RoboDK station: Robot_2TCP.rdk

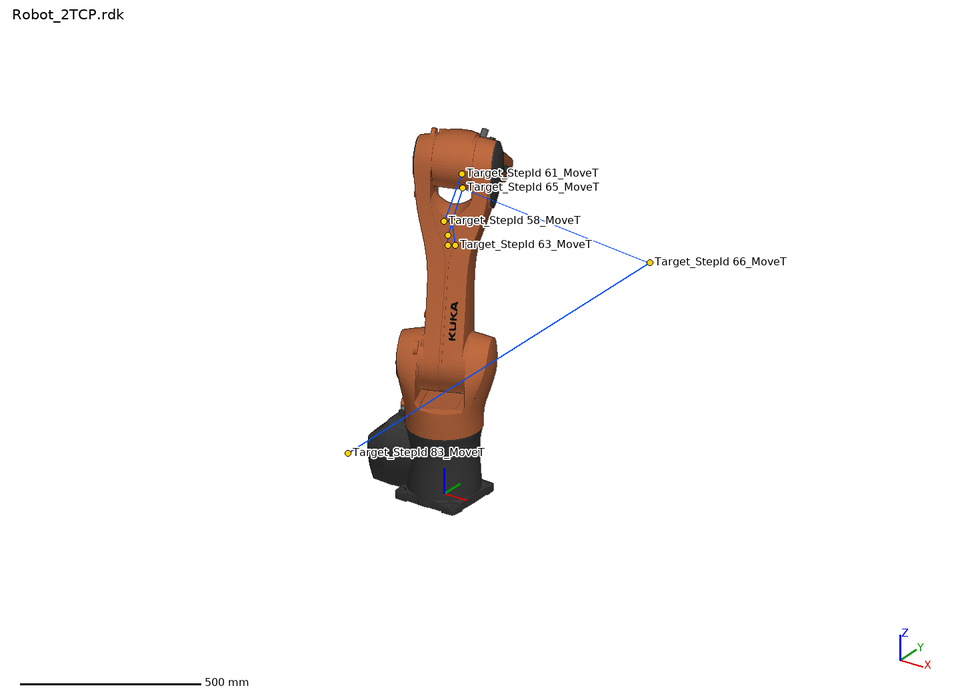
[picture v0: the station drawn from its stored meshes, robots at their saved joint values, targets as dots, program paths as lines]
Station Robot_2TCP (saved by RoboDK 5.1.0). Poses are relative to the parent item; angles as X-Y-Z fixed-axis rotations.
  - frame KUKA KR 10 R1100 sixx Base at (0, 0, 0) mm
    - robot KUKA KR 10 R1100 sixx: 6 axes, payload 10 kg, reach 1101 mm, repeatability 0.03 mm, weight 54 kg
        modified DH rows (alpha deg, a mm, theta deg, d mm): 0, 0, 0, 400; -90, 25, 0, 0; 0, 560, -90, 0; -90, 35, 0, 515; 90, 0, 0, 0; -90, 0, 180, 80
        joint limits [-170, -190, -120, -185, -120, -350] to [170, 45, 156, 185, 120, 350]; home [0, -90, 90, 0, 0, 0]; saved at [-113.458, -74.372, 105.005, -12.718, 115.702, 149.13]
      - tool Greifer1, TCP at (43.5, -78.7, 129.7) mm, rotated rx 90 ry 0 rz 0 deg
      - tool Greifer2, TCP at (40, 0, 186.7) mm
    - target Target_StepId 61_MoveType.Joint (joint target) at (-247.75, 438.18, 739.43) mm, rotated rx -105.36 ry -9.62 rz 92.45 deg; joints [-121.962, -102.168, 105.538, 18.09, 86.239, 148.055] of KUKA KR 10 R1100 sixx
    - target Target_StepId 58_MoveType.Frame (Cartesian target) at (-307.35, 439.57, 576.8) mm, rotated rx -105.36 ry -9.62 rz 92.45 deg; joints [-128.201, -95.591, 118.458, 19.243, 69.676, 135.809] of KUKA KR 10 R1100 sixx
    - target Target_StepId 62_MoveType.Frame (Cartesian target) at (-282.44, 439.49, 583.54) mm, rotated rx -105.36 ry -9.62 rz 92.45 deg; joints [-125.678, -97.441, 119.28, 19.266, 69.877, 138.518] of KUKA KR 10 R1100 sixx
    - target Target_StepId 63_MoveType.Frame (Cartesian target) at (-267.1, 434.01, 516.13) mm, rotated rx -115.88 ry 53.49 rz 68.75 deg; joints [-111.554, -74.002, 107.434, -10.728, 113.29, 151.492] of KUKA KR 10 R1100 sixx
    - target Target_StepId 60_MoveType.Frame (Cartesian target) at (-292.02, 433.98, 509.43) mm, rotated rx -115.88 ry 53.49 rz 68.75 deg; joints [-113.636, -72.782, 106.634, -12.563, 112.528, 149.741] of KUKA KR 10 R1100 sixx
    - target Target_StepId 64_MoveType.Frame (Cartesian target) at (-289.75, 433.74, 539.34) mm, rotated rx -115.88 ry 53.49 rz 68.75 deg; joints [-113.458, -74.372, 105.005, -12.718, 115.702, 149.13] of KUKA KR 10 R1100 sixx
    - target Target_StepId 65_MoveType.Frame (Cartesian target) at (-239.81, 432.38, 699.35) mm, rotated rx -115.88 ry 53.49 rz 68.75 deg; joints [0, -90, 90, 0, 0, 0] of KUKA KR 10 R1100 sixx
    - target Target_StepId 66_MoveType.Joint (joint target) at (749.7, -78.7, 951.5) mm, rotated rx 0 ry 90 rz -90 deg; joints [0, 0, 0, 0, 0, 0] of KUKA KR 10 R1100 sixx
    - target Target_StepId 81_MoveType.Joint (joint target) at (749.7, -78.7, 951.5) mm, rotated rx 0 ry 90 rz -90 deg; joints [79.238, -54.626, 102.86, -115.621, 68.886, -126.912] of KUKA KR 10 R1100 sixx
    - target Target_StepId 83_MoveType.Frame (Cartesian target) at (312.31, -910.02, 574.5) mm, rotated rx 0 ry 0 rz -111.98 deg; joints [80.378, -48.158, 90.554, 67.471, -67.234, 46.988] of KUKA KR 10 R1100 sixx
  - program Prg (40 instructions, listed below)
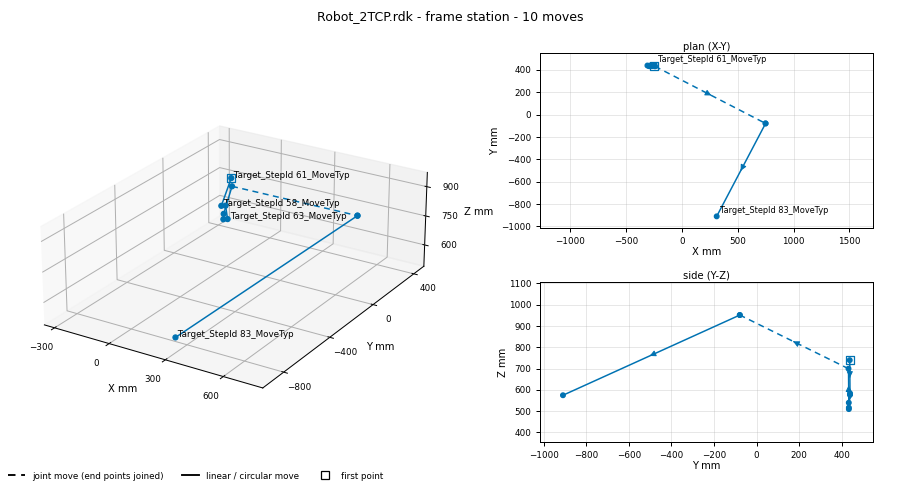
[picture p0: tool path of Robot_2TCP.rdk in frame station, 10 of 10 moves have a stored position in this frame; points joined in program order, loops and branches not executed]

--- program Prg (robot KUKA KR 10 R1100 sixx) ---
  Set Tool: Greifer1
  Smooth(10)
  Set speed (225.0 deg/s)
  MoveJ (Target_StepId 61_MoveType.Joint)
  Set Tool: Greifer1
  Smooth(0)
  Set speed (2000.0 mm/s)
  MoveL (Target_StepId 58_MoveType.Frame)
  Set Tool: Greifer1
  Smooth(10)
  Set speed (2000.0 mm/s)
  MoveL (Target_StepId 62_MoveType.Frame)
  Set Tool: Greifer1
  Smooth(10)
  Set speed (2000.0 mm/s)
  MoveL (Target_StepId 63_MoveType.Frame)
  Set Tool: Greifer1
  Smooth(0)
  Set speed (2000.0 mm/s)
  MoveL (Target_StepId 60_MoveType.Frame)
  Set Tool: Greifer1
  Smooth(10)
  Set speed (2000.0 mm/s)
  MoveL (Target_StepId 64_MoveType.Frame)
  Set Tool: Greifer1
  Smooth(10)
  Set speed (2000.0 mm/s)
  MoveL (Target_StepId 65_MoveType.Frame)
  Set Tool: Greifer1
  Smooth(10)
  Set speed (225.0 deg/s)
  MoveJ (Target_StepId 66_MoveType.Joint)
  Set Tool: Greifer1
  Smooth(10)
  Set speed (225.0 deg/s)
  MoveJ (Target_StepId 81_MoveType.Joint)
  Set Tool: Greifer1
  Smooth(1)
  Set speed (2000.0 mm/s)
  MoveL (Target_StepId 83_MoveType.Frame)
